PROGRAM SafetyPLC
VAR

(*=========================		SAFETY PLC		==========================*)	



(*========================================================================*)

END_VAR

(*=========================		SAFETY PLC		==========================*)



(*========================================================================*)

END_PROGRAM

(* stored: Version 1.1.0.1, ProductVersion 3.1.4024.11
   POU SafetyPLC: Id {d72391e9-50f0-4b14-82db-156d9d838551}, SpecialFunc None *)
